TYPE DUT_Test_1 :
STRUCT
	a : BOOL;
	b : REAL;
	c : string(200);
END_STRUCT
END_TYPE

(* stored: Version 1.1.0.1, ProductVersion 3.1.4024.11
   DUT DUT_Test_1: Id {acd52f52-0eb1-4843-96ea-cff538cf5b76} *)
